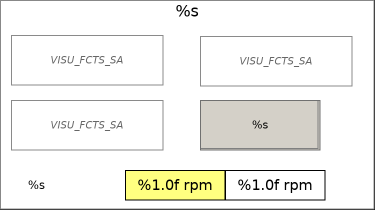
VISUALIZATION SA_ROT  // 375x210
VAR_IN_OUT
	m_Input_ROT:				BLOCK_ROTATION_CONTINUE_ATV;
	m_Input_PRG:				BLOCK_PRG_MOUVEMENT_PS;
END_VAR
    Rectangle (0,0 375x210), "%s", text list: 'TextList_Type_Moteur', text index: 1
    Button (200,100 120x50), "%s", input disabled if: not PRG_USER.ACTU_USER.FONCTION_SA, text list: 'TextList_Basiques', text index: 19
        tap m_Input_ROT.CO_Modif
    RoundedRectangle (125,170 100x30), "%1.0f rpm", text variable: m_Input_ROT.PRM_vitesse, input disabled if: (NOT PRG_User.ACTU_USER.MAINTENANCE AND NOT PRG_User.ACTU_USER.FONCTION_SA AND NOT PRG_User.ACTU_USER.MODIF_ENLIGNE) OR ( MACHINE.STATE_Manu )
        OnMouseDown: write the text variable via InputWithLimits, min m_Input_ROT.CONF_VMIN, max m_Input_ROT.CONF_VMAX, title 'Speed'
    Rectangle (25,170 100x30), "%s", text list: 'TextList_Moteurs', text index: 7
    RoundedRectangle (225,170 100x30), "%1.0f rpm", text variable: m_Input_ROT.STATE_Vitesse
    Frame (11,35 152x50), invisible if: not m_Input_PRG.CONF_Rotation
        shows VISU_FCTS_SA(m_Input_ID_XML := 15, m_Input_Operation := m_Input_ROT.OP_ROTATION, m_Input_UserRight := PRG_USER.ACTU_USER.FONCTION_SA AND NOT MACHINE.STATE_Prod)
        p768090162: m_Input_ROT.OP_ROTATION
        p1726406813: PRG_USER.ACTU_USER.FONCTION_SA AND NOT MACHINE.STATE_Prod
    Frame (200,36 152x50)
        shows VISU_FCTS_SA(m_Input_ID_XML := 7, m_Input_Operation := m_Input_ROT.OP_ARRET, m_Input_UserRight := PRG_USER.ACTU_USER.FONCTION_SA AND NOT MACHINE.STATE_Prod)
        p768090162: m_Input_ROT.OP_ARRET
        p1726406813: PRG_USER.ACTU_USER.FONCTION_SA AND NOT MACHINE.STATE_Prod
    Frame (11,100 152x50), invisible if: not m_Input_PRG.CONF_Positionnement
        shows VISU_FCTS_SA(m_Input_ID_XML := 8, m_Input_Operation := m_Input_ROT.OP_POSITION, m_Input_UserRight := PRG_USER.ACTU_USER.FONCTION_SA AND NOT MACHINE.STATE_Prod)
        p768090162: m_Input_ROT.OP_POSITION
        p1726406813: PRG_USER.ACTU_USER.FONCTION_SA AND NOT MACHINE.STATE_Prod
END_VISUALIZATION

(* stored: Version 1.1.0.1, ProductVersion 3.1.4024.12
   Visu SA_ROT: Id {4587ad4f-10b0-4928-8b47-4478c1dffcae} *)
